// TIA Portal V20 export
// export: Created 2026-07-10T11:12:22.8829142Z, ExportSetting WithDefaults, DisplayName Totally Integrated Automation Portal, DisplayVersion V20, DisplayName TIA Portal Openness, DisplayVersion V20, DisplayName TIA Portal Version Control Interface, DisplayVersion V20, DisplayName STEP 7 Professional, DisplayVersion V20, DisplayName STEP 7 Safety, DisplayVersion V20, DisplayName WinCC Basic/Comfort/Advanced, DisplayVersion V20, DisplayName WinCC Unified, DisplayVersion V20
FUNCTION_BLOCK "AIHandler"   // FB3, SCL
{ S7_Optimized_Access := 'TRUE' }
VERSION : 0.1
// stored: AutoNumber true, IsIECCheckEnabled false, IsRetainMemResEnabled false, MemoryReserve 100, SetENOAutomatically false, UDAEnableTagReadback false
   VAR_INPUT
      Value : Real;
      ValueMin : Real;
      ValueMax : Real;
      ValueOffset : Real;
      OutputMin : Real;
      OutputMax : Real;
      TimeBase : Time := T#1s;
   END_VAR
   VAR_OUTPUT
      Output : Real;
      Error : Bool;
   END_VAR
   VAR
      ConvertedValue : Real;
      TON1 { S7_SetPoint := 'True'} : TON_TIME;
      DelayTON { S7_SetPoint := 'True'} : TON_TIME;
      FilterArray : Array[0..199] of Real;
      FilterTime : Time;
      i : Int;
      sum : Real;
      FilteredValue : Real;
      one : Bool;
   END_VAR
   VAR CONSTANT
      TimeDelay : Time := T#120s;
   END_VAR
BEGIN

   #FilterTime := #TimeBase * 1000 /50;

   #DelayTON(IN := TRUE,
             PT := #FilterTime);


   IF #DelayTON.Q = TRUE THEN
           RESET_TIMER(#DelayTON);
           #sum := #sum + #Value;
           #i := #i + 1;
           IF (#i >= 50) THEN
               #i := 0;
               #FilteredValue := #sum / 50.0;
               #ConvertedValue := (#FilteredValue - #ValueMin) / (#ValueMax - #ValueMin) * (#OutputMax - #OutputMin) + #OutputMin;
               #sum := 0;
               IF (#ConvertedValue < 0) THEN
                   #Output := 0;
               ELSE
                   #Output := #ConvertedValue + #ValueOffset;
               END_IF;
           END_IF;
   END_IF;

   #TON1(IN := #Value > 30000,
         PT := #TimeDelay,
         Q => #Error);
END_FUNCTION_BLOCK
